FUNCTION_BLOCK ThisXTS EXTENDS Xts
VAR
END_VAR

METHOD MoverHomeSequence : BOOL
VAR
	i : INT;
END_VAR
FOR i := 0 TO 7 DO 
	_MoverArray[i].MoveTo(600.0,1000.0,FALSE);
END_FOR
END_METHOD

END_FUNCTION_BLOCK

(* stored: Version 1.1.0.1, ProductVersion 3.1.4026.12
   POU ThisXTS: Id {adc628a7-7a2e-4111-937d-b66eb159493c}, SpecialFunc None
   Method MoverHomeSequence: Id {dd65f3ed-d01b-4f9f-95cc-8438905256ec} *)
